{attribute 'GeneratedUsingTerminal: EL3783-0000-0018'}
{attribute addProperty BoxType "EL3783-0000-0018"}
{attribute addProperty Id "ARRAY_0INT2ARRAY_1INT2ARRAY_2INT2ARRAY_3INT2ARRAY_4INT2ARRAY_5INT2ARRAY_6INT2ARRAY_7INT2ARRAY_8INT2ARRAY_9INT2ARRAY_10INT2ARRAY_11INT2ARRAY_12INT2ARRAY_13INT2ARRAY_14INT2ARRAY_15INT2ARRAY_16INT2ARRAY_17INT2ARRAY_18INT2ARRAY_19INT2"}
{attribute addProperty CRC "285858986"}
{attribute addProperty Size "40"}
TYPE U2_Samples_1109DCAA :
STRUCT
	{attribute addProperty Name "ARRAY_0"}
	ARRAY_0 : INT;
	{attribute addProperty Name "ARRAY_1"}
	ARRAY_1 : INT;
	{attribute addProperty Name "ARRAY_2"}
	ARRAY_2 : INT;
	{attribute addProperty Name "ARRAY_3"}
	ARRAY_3 : INT;
	{attribute addProperty Name "ARRAY_4"}
	ARRAY_4 : INT;
	{attribute addProperty Name "ARRAY_5"}
	ARRAY_5 : INT;
	{attribute addProperty Name "ARRAY_6"}
	ARRAY_6 : INT;
	{attribute addProperty Name "ARRAY_7"}
	ARRAY_7 : INT;
	{attribute addProperty Name "ARRAY_8"}
	ARRAY_8 : INT;
	{attribute addProperty Name "ARRAY_9"}
	ARRAY_9 : INT;
	{attribute addProperty Name "ARRAY_10"}
	ARRAY_10 : INT;
	{attribute addProperty Name "ARRAY_11"}
	ARRAY_11 : INT;
	{attribute addProperty Name "ARRAY_12"}
	ARRAY_12 : INT;
	{attribute addProperty Name "ARRAY_13"}
	ARRAY_13 : INT;
	{attribute addProperty Name "ARRAY_14"}
	ARRAY_14 : INT;
	{attribute addProperty Name "ARRAY_15"}
	ARRAY_15 : INT;
	{attribute addProperty Name "ARRAY_16"}
	ARRAY_16 : INT;
	{attribute addProperty Name "ARRAY_17"}
	ARRAY_17 : INT;
	{attribute addProperty Name "ARRAY_18"}
	ARRAY_18 : INT;
	{attribute addProperty Name "ARRAY_19"}
	ARRAY_19 : INT;
END_STRUCT
END_TYPE

(* stored: Version 1.2.0.0, ProductVersion 3.1.4024.9
   DUT U2_Samples_1109DCAA: Id {6fc5eb4b-6171-4e76-be9e-febe75abeeab} *)
